// TIA Portal project "Sistema_semaforico3" (V15.1)

(* hardware
DEVICE "S7-1200 station_1"  S7-1200 Station
   slot 0: "Telaio di montaggio_0"  S7-1200 Rack  Rack  V1.0
   slot 1: "PLC_1"  CPU 1214C DC/DC/DC  6ES7 214-1AG40-0XB0  V4.2
*)

// ===== PLC "PLC_1"  CPU 1214C DC/DC/DC =====

VAR_GLOBAL   // PLC tag table "Tabella delle variabili standard"
   "P" AT %I0.0 : Bool;
   "prenotato" AT %Q0.0 : Bool;
   "start" AT %I0.1 : Bool;
END_VAR

VAR_GLOBAL CONSTANT   // PLC tag table "Tabella delle variabili standard"
   "tempoVerde" : Time := T#55s;
   "tempoGiallo" : Time := T#5s;
   "tempoRosso" : Time := T#60s;
END_VAR

DATA_BLOCK "variabili_stato"   // DB1
{ S7_Optimized_Access := 'TRUE' }
VERSION : 0.1
   VAR RETAIN
      home : Bool := true;
      VR : Bool;
      GR : Bool;
      RV : Bool;
      RG : Bool;
      RR : Bool;
   END_VAR
BEGIN
END_DATA_BLOCK

// folder: System blocks/Program resources

DATA_BLOCK "IEC_Timer_0_DB"   // DB2
{ S7_Optimized_Access := 'TRUE' }
AUTHOR : Simatic
FAMILY : IEC
NAME : IEC_TMR
VERSION : 1.0
// stored: InstanceOfName IEC_TIMER
"IEC_TIMER"
BEGIN
END_DATA_BLOCK

DATA_BLOCK "IEC_Timer_0_DB_1"   // DB3
{ S7_Optimized_Access := 'TRUE' }
AUTHOR : Simatic
FAMILY : IEC
NAME : IEC_TMR
VERSION : 1.0
// stored: InstanceOfName IEC_TIMER
"IEC_TIMER"
BEGIN
END_DATA_BLOCK

DATA_BLOCK "IEC_Timer_0_DB_2"   // DB4
{ S7_Optimized_Access := 'TRUE' }
AUTHOR : Simatic
FAMILY : IEC
NAME : IEC_TMR
VERSION : 1.0
// stored: InstanceOfName IEC_TIMER
"IEC_TIMER"
BEGIN
END_DATA_BLOCK

DATA_BLOCK "IEC_Timer_0_DB_3"   // DB5
{ S7_Optimized_Access := 'TRUE' }
AUTHOR : Simatic
FAMILY : IEC
NAME : IEC_TMR
VERSION : 1.0
// stored: InstanceOfName IEC_TIMER
"IEC_TIMER"
BEGIN
END_DATA_BLOCK

DATA_BLOCK "IEC_Timer_0_DB_4"   // DB6
{ S7_Optimized_Access := 'TRUE' }
AUTHOR : Simatic
FAMILY : IEC
NAME : IEC_TMR
VERSION : 1.0
// stored: InstanceOfName IEC_TIMER
"IEC_TIMER"
BEGIN
END_DATA_BLOCK

// folder: (top level)

ORGANIZATION_BLOCK "Main"   // OB1, LAD, ProgramCycle
TITLE = "Main Program Sweep (Cycle)"
{ S7_Optimized_Access := 'TRUE' }
VERSION : 0.1
   VAR_INPUT
      Initial_Call : Bool;   // Initial call of this OB
      Remanence : Bool;   // =True, if remanent data are available
   END_VAR
   VAR_TEMP   // added for the SCL form of the ladder/FBD networks
      _w1 : Bool;
   END_VAR
BEGIN

REGION Network 1
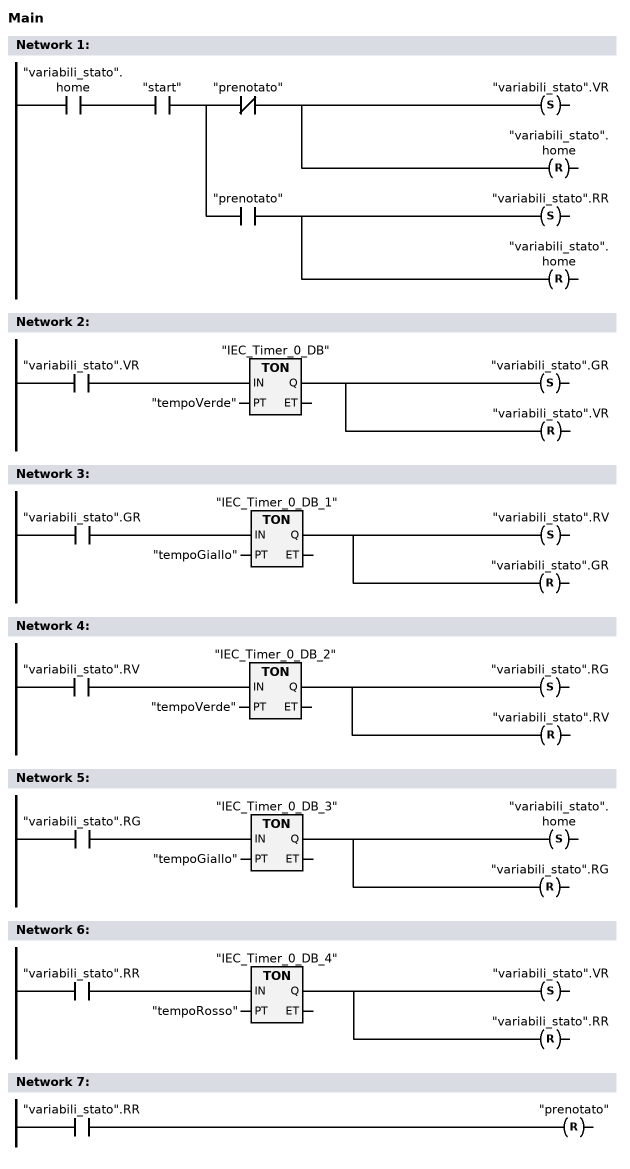
   RUNG wire#powerrail
      Contact( "variabili_stato".home )
      Contact( "start" )
      wire#w1
      I_Contact( "prenotato" )
      wire#w2
      S_Coil( "variabili_stato".VR )
   END_RUNG
   RUNG wire#w2
      R_Coil( "variabili_stato".home )
   END_RUNG
   RUNG wire#w1
      Contact( "prenotato" )
      wire#w3
      S_Coil( "variabili_stato".RR )
   END_RUNG
   RUNG wire#w3
      R_Coil( "variabili_stato".home )
   END_RUNG
   // the same network as SCL:
   #_w1 := "variabili_stato".home AND "start";
   IF #_w1 AND NOT "prenotato" THEN
       "variabili_stato".VR := TRUE;
       "variabili_stato".home := FALSE;
   END_IF;
   IF #_w1 AND "prenotato" THEN
       "variabili_stato".RR := TRUE;
       "variabili_stato".home := FALSE;
   END_IF;
END_REGION

REGION Network 2
   "IEC_Timer_0_DB".TON(IN := "variabili_stato".VR, PT := "tempoVerde");
   IF "IEC_Timer_0_DB".Q THEN
       "variabili_stato".GR := TRUE;
       "variabili_stato".VR := FALSE;
   END_IF;
END_REGION

REGION Network 3
   "IEC_Timer_0_DB_1".TON(IN := "variabili_stato".GR, PT := "tempoGiallo");
   IF "IEC_Timer_0_DB_1".Q THEN
       "variabili_stato".RV := TRUE;
       "variabili_stato".GR := FALSE;
   END_IF;
END_REGION

REGION Network 4
   "IEC_Timer_0_DB_2".TON(IN := "variabili_stato".RV, PT := "tempoVerde");
   IF "IEC_Timer_0_DB_2".Q THEN
       "variabili_stato".RG := TRUE;
       "variabili_stato".RV := FALSE;
   END_IF;
END_REGION

REGION Network 5
   "IEC_Timer_0_DB_3".TON(IN := "variabili_stato".RG, PT := "tempoGiallo");
   IF "IEC_Timer_0_DB_3".Q THEN
       "variabili_stato".home := TRUE;
       "variabili_stato".RG := FALSE;
   END_IF;
END_REGION

REGION Network 6
   "IEC_Timer_0_DB_4".TON(IN := "variabili_stato".RR, PT := "tempoRosso");
   IF "IEC_Timer_0_DB_4".Q THEN
       "variabili_stato".VR := TRUE;
       "variabili_stato".RR := FALSE;
   END_IF;
END_REGION

REGION Network 7
   RUNG wire#powerrail
      Contact( "variabili_stato".RR )
      R_Coil( "prenotato" )
   END_RUNG
   // the same network as SCL:
   IF "variabili_stato".RR THEN "prenotato" := FALSE; END_IF;
END_REGION
END_ORGANIZATION_BLOCK

ORGANIZATION_BLOCK "Hardware interrupt"   // OB40, LAD, HWProcessInterrupt
{ S7_Optimized_Access := 'TRUE' }
VERSION : 0.1
   VAR_INPUT
      LADDR : Hw_Io;   // Hardware identifier
      USI : Word;   // User structure identifier
      IChannel : USInt;   // Interrupt channel number
      EventType : Byte;   // EventType
   END_VAR
BEGIN

REGION Network 1
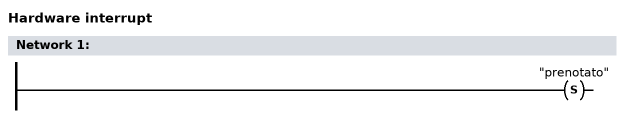
   RUNG wire#powerrail
      S_Coil( "prenotato" )
   END_RUNG
   // the same network as SCL:
   "prenotato" := TRUE;
END_REGION
END_ORGANIZATION_BLOCK